(* PLC project op_alarm, Dassault Systèmes ControlBuild 2024x *)
(* stored: creationDateTime 2023-10-03T11:13:50-01:00 *)

FUNCTION_BLOCK tni_train.op_alarm
  VAR_INPUT
    enableAlarm : BOOL := false;
    resetKey : BOOL := false;
  END_VAR
  VAR_OUTPUT
    alarm : BOOL := false;
  END_VAR
  VAR
    i_rs1 : DINT := 0;
  END_VAR

(* LD diagram, written out as Structured Text *)
1:
rs1(S := enableAlarm, R1 := resetKey);
alarm := rs1.Q1;
END_FUNCTION_BLOCK
